PROGRAM MAIN_LD
VAR	

	// ========= System Control / FSM Variables =========
	
	MainCommands 		: MainCommands_typ; 		// command struct for cycling thru the state machine
	MainState    		: MainStateMachine_enum;   	// enumeration for the Main state machine
	System				: Mediator;					// System-level control object

	// ========= Linked NC Variables & References =========
	
	Mover    			: ARRAY[1..GVL.NUM_MOVERS] OF Mover; 	// instantiation of Mover objects. Matches the number of movers on the system
	
	// ========= Objectives & Parameters =========

	ParameterSet		: MotionParameters_typ;
	
	MoverList			: ARRAY[0..GVL.NUM_MOVERLISTS-1] OF MoverList;
	PositionTrigger		: ARRAY[0..GVL.NUM_POSITIONTRIGGERS-1] OF PositionTrigger;
	Station				: ARRAY[0..GVL.NUM_STATIONS-1] OF Station;
	Track				: ARRAY[0..GVL.NUM_TRACKS] OF Track;
	Zone				: ARRAY[0..GVL.NUM_ZONES-1] OF Zone;
	
    // ========= Helper, State, & Index Variables =========
	
    i                	: UINT; 	// index variable; gets reused in various FOR loops
    n                	: UINT; 	// secondary index variable, for enabling movers
	
	// ========= Example Application Variables =========

    nextStation 			: USINT := 4;
                    	
    lowVelocity    			: LREAL := 200;  	// mm/s
    mediumVelocity 			: LREAL := 800;  	// mm/s
    highVelocity   			: LREAL := 1200; 	// mm/s
	
	StationTimer 			: ARRAY[0..GVL.NUM_STATIONS] OF TON; // timer blocks, for station dwells
	InitialParameterSet		: MotionParameters_typ;
	
	// ========= Additional Ladder Variables =========
	MS_Disabled						: BOOL;
	MS_Initializing					: BOOL;
	MS_Enabled						: BOOL;
	MS_Run							: BOOL;
	MS_Stopping						: BOOL;
	MS_Stopped						: BOOL;
	MS_Disabling					: BOOL;
	MS_Error						: BOOL;
	MS_Debug						: BOOL;
	
	MS_Enabled_StartReady			: BOOL;
	StationGroupInPosition			: BOOL;
	StationGroupMoversInPosition	: BOOL;
	Station1_TimerIn: BOOL;
END_VAR
VAR // added by the converter: edge detectors and wires of the graphical bodies
    _w1, _w2, _w3, _w4, _w5, _w6, _w7, _w8, _w9 : BOOL;
END_VAR

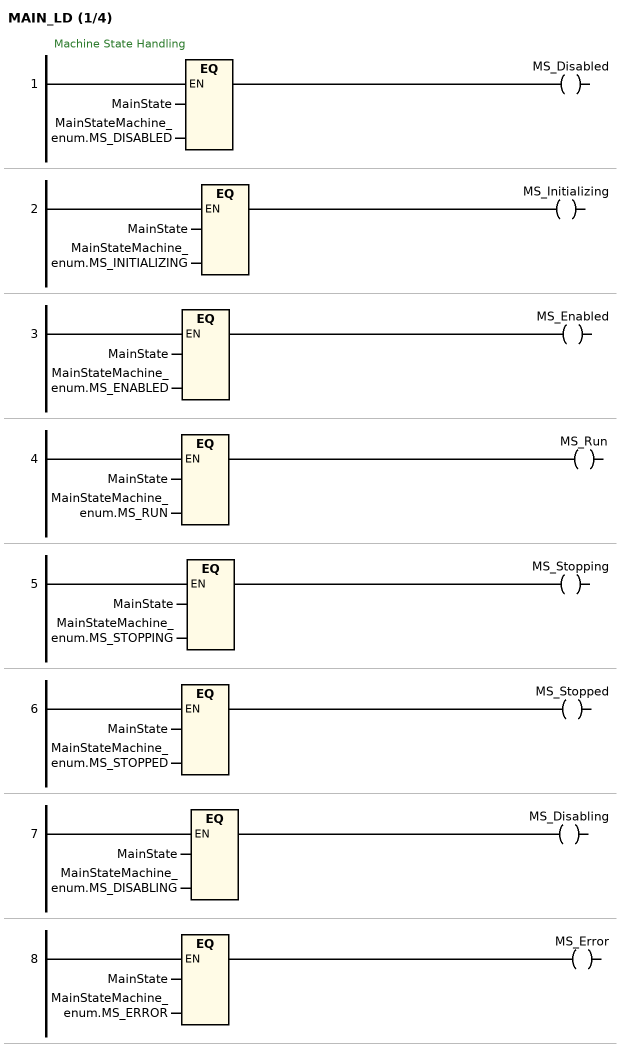
// NETWORK 1
// Machine State Handling
MS_Disabled := MainState = MainStateMachine_enum.MS_DISABLED;

// NETWORK 2
MS_Initializing := MainState = MainStateMachine_enum.MS_INITIALIZING;

// NETWORK 3
MS_Enabled := MainState = MainStateMachine_enum.MS_ENABLED;

// NETWORK 4
MS_Run := MainState = MainStateMachine_enum.MS_RUN;

// NETWORK 5
MS_Stopping := MainState = MainStateMachine_enum.MS_STOPPING;

// NETWORK 6
MS_Stopped := MainState = MainStateMachine_enum.MS_STOPPED;

// NETWORK 7
MS_Disabling := MainState = MainStateMachine_enum.MS_DISABLING;

// NETWORK 8
MS_Error := MainState = MainStateMachine_enum.MS_ERROR;

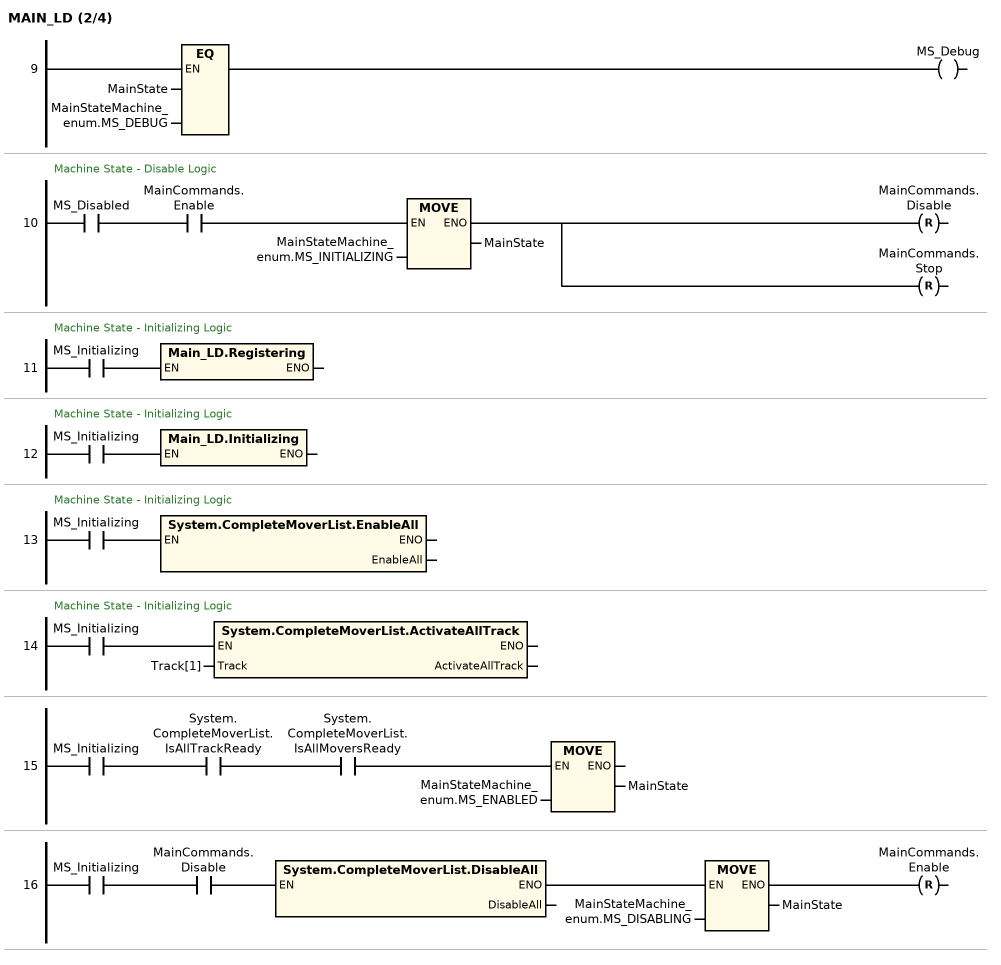
// NETWORK 9
MS_Debug := MainState = MainStateMachine_enum.MS_DEBUG;

// NETWORK 10
// Machine State - Disable Logic
_w1 := MS_Disabled AND MainCommands.Enable;
IF _w1 THEN MainState := MainStateMachine_enum.MS_INITIALIZING; END_IF
MainCommands.Disable R= _w1;
MainCommands.Stop R= _w1;

// NETWORK 11
// Machine State - Initializing Logic
IF MS_Initializing THEN Main_LD.Registering(); END_IF

// NETWORK 12
// Machine State - Initializing Logic
IF MS_Initializing THEN Main_LD.Initializing(); END_IF

// NETWORK 13
// Machine State - Initializing Logic
IF MS_Initializing THEN System.CompleteMoverList.EnableAll(); END_IF

// NETWORK 14
// Machine State - Initializing Logic
IF MS_Initializing THEN System.CompleteMoverList.ActivateAllTrack(Track := Track[1]); END_IF

// NETWORK 15
IF MS_Initializing AND System.CompleteMoverList.IsAllTrackReady AND System.CompleteMoverList.IsAllMoversReady THEN
    MainState := MainStateMachine_enum.MS_ENABLED;
END_IF

// NETWORK 16
_w2 := MS_Initializing AND MainCommands.Disable;
IF _w2 THEN System.CompleteMoverList.DisableAll(); END_IF
IF _w2 THEN MainState := MainStateMachine_enum.MS_DISABLING; END_IF
MainCommands.Enable R= _w2;

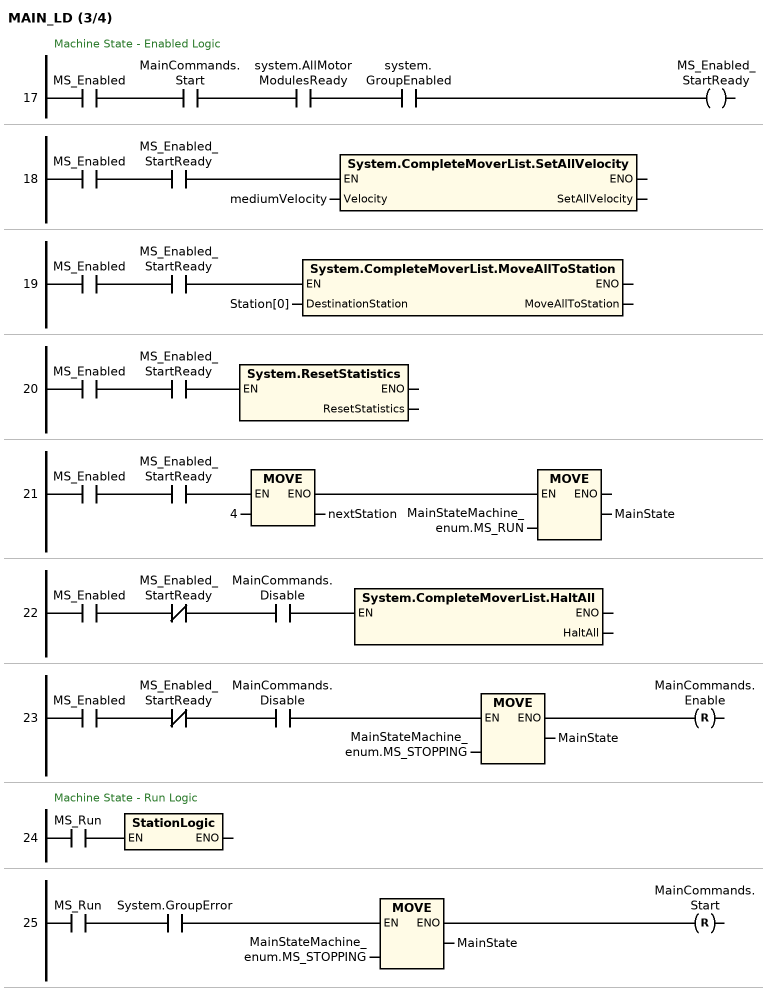
// NETWORK 17
// Machine State - Enabled Logic
MS_Enabled_StartReady := MS_Enabled AND MainCommands.Start AND system.AllMotorModulesReady AND system.GroupEnabled;

// NETWORK 18
IF MS_Enabled AND MS_Enabled_StartReady THEN
    System.CompleteMoverList.SetAllVelocity(Velocity := mediumVelocity);
END_IF

// NETWORK 19
IF MS_Enabled AND MS_Enabled_StartReady THEN
    System.CompleteMoverList.MoveAllToStation(DestinationStation := Station[0]);
END_IF

// NETWORK 20
IF MS_Enabled AND MS_Enabled_StartReady THEN System.ResetStatistics(); END_IF

// NETWORK 21
_w3 := MS_Enabled AND MS_Enabled_StartReady;
IF _w3 THEN nextStation := 4; END_IF
IF _w3 THEN MainState := MainStateMachine_enum.MS_RUN; END_IF

// NETWORK 22
IF MS_Enabled AND NOT MS_Enabled_StartReady AND MainCommands.Disable THEN
    System.CompleteMoverList.HaltAll();
END_IF

// NETWORK 23
_w4 := MS_Enabled AND NOT MS_Enabled_StartReady AND MainCommands.Disable;
IF _w4 THEN MainState := MainStateMachine_enum.MS_STOPPING; END_IF
MainCommands.Enable R= _w4;

// NETWORK 24
// Machine State - Run Logic
IF MS_Run THEN StationLogic(); END_IF

// NETWORK 25
_w5 := MS_Run AND System.GroupError;
IF _w5 THEN MainState := MainStateMachine_enum.MS_STOPPING; END_IF
MainCommands.Start R= _w5;

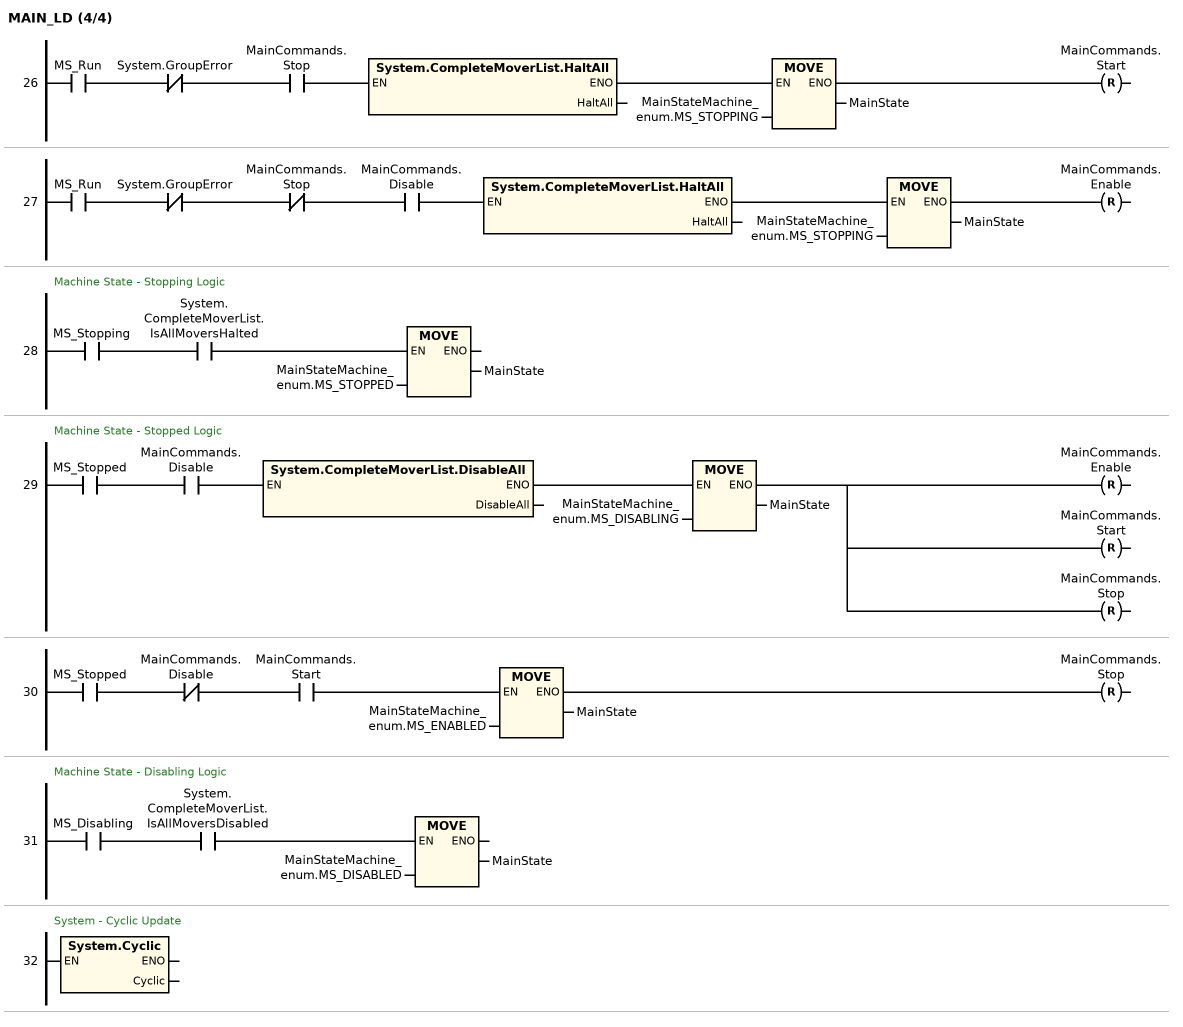
// NETWORK 26
_w6 := MS_Run AND NOT System.GroupError AND MainCommands.Stop;
IF _w6 THEN System.CompleteMoverList.HaltAll(); END_IF
IF _w6 THEN MainState := MainStateMachine_enum.MS_STOPPING; END_IF
MainCommands.Start R= _w6;

// NETWORK 27
_w7 := MS_Run AND NOT System.GroupError AND NOT MainCommands.Stop AND MainCommands.Disable;
IF _w7 THEN System.CompleteMoverList.HaltAll(); END_IF
IF _w7 THEN MainState := MainStateMachine_enum.MS_STOPPING; END_IF
MainCommands.Enable R= _w7;

// NETWORK 28
// Machine State - Stopping Logic
IF MS_Stopping AND System.CompleteMoverList.IsAllMoversHalted THEN
    MainState := MainStateMachine_enum.MS_STOPPED;
END_IF

// NETWORK 29
// Machine State - Stopped Logic
_w8 := MS_Stopped AND MainCommands.Disable;
IF _w8 THEN System.CompleteMoverList.DisableAll(); END_IF
IF _w8 THEN MainState := MainStateMachine_enum.MS_DISABLING; END_IF
MainCommands.Enable R= _w8;
MainCommands.Start R= _w8;
MainCommands.Stop R= _w8;

// NETWORK 30
_w9 := MS_Stopped AND NOT MainCommands.Disable AND MainCommands.Start;
IF _w9 THEN MainState := MainStateMachine_enum.MS_ENABLED; END_IF
MainCommands.Stop R= _w9;

// NETWORK 31
// Machine State - Disabling Logic
IF MS_Disabling AND System.CompleteMoverList.IsAllMoversDisabled THEN
    MainState := MainStateMachine_enum.MS_DISABLED;
END_IF

// NETWORK 32
// System - Cyclic Update
System.Cyclic();

ACTION Initializing:


	// Initialize station positions
	Station[0].Position 		:= 5;
	Station[1].Position 		:= 750;
	Station[2].Position 		:= 1200;
	Station[3].Position 		:= 1300;
	Station[4].Position 		:= 1400;

	PositionTrigger[0].Position := 1500;
	PositionTrigger[1].Position := 2000;
	PositionTrigger[2].Position := 3500;

	Zone[0].StartPosition		:= 3750;
	Zone[0].EndPosition   		:= 750;

	Zone[1].StartPosition 		:= 750;
	Zone[1].EndPosition   		:= 1750;

	Zone[2].StartPosition 		:= 1750;
	Zone[2].EndPosition   		:= 2750;

	Zone[3].StartPosition		:= 2750;
	Zone[3].EndPosition   		:= 3750;

	InitialParameterSet.Velocity		:= 1000;		// mm/s
	InitialParameterSet.Acceleration	:= 10_000;		// mm/s2
	InitialParameterSet.Deceleration	:= 10_000;		// mm/s2
	InitialParameterSet.Jerk			:= 100_000;		// mm/s3
	InitialParameterSet.Gap				:= 85;			// mm
	InitialParameterSet.Direction		:= mcDirectionPositive;	
	
	System.CompleteMoverList.ApplyAllParameterSet( InitialParameterSet );
END_ACTION

ACTION Registering:
	

		// Add all Movers to the Mediator
		FOR i := 1 TO GVL.NUM_MOVERS DO
			System.AddMover( Mover[i] );
		END_FOR
	
		// Add all Mover Lists to the Mediator
		FOR i := 0 TO GVL.NUM_MOVERLISTS - 1 DO
			System.AddMoverList( MoverList[i] );
		END_FOR
		
		// Add all PositionTriggers to the Mediator
		FOR i := 0 TO GVL.NUM_POSITIONTRIGGERS - 1 DO
			System.AddPositionTrigger( PositionTrigger[i] );
		END_FOR
		
		// Add all Stations to the Mediator
		FOR i := 0 TO GVL.NUM_STATIONS - 1 DO
			System.AddStation( Station[i] );
		END_FOR
		
		// Add all Tracks to the Mediator
		// note track zero is a special case, so the loop is one larger than the rest of the initalization loops
		FOR i := 0 TO GVL.NUM_TRACKS DO
			Track[i].Id := UINT_TO_INT(i);
			System.AddTrack( Track[i] );
		END_FOR
		
		// Add all Zones to the Mediator
		FOR i := 0 TO GVL.NUM_ZONES - 1 DO
			System.AddZone( Zone[i] );
		END_FOR
END_ACTION

ACTION StationLogic:
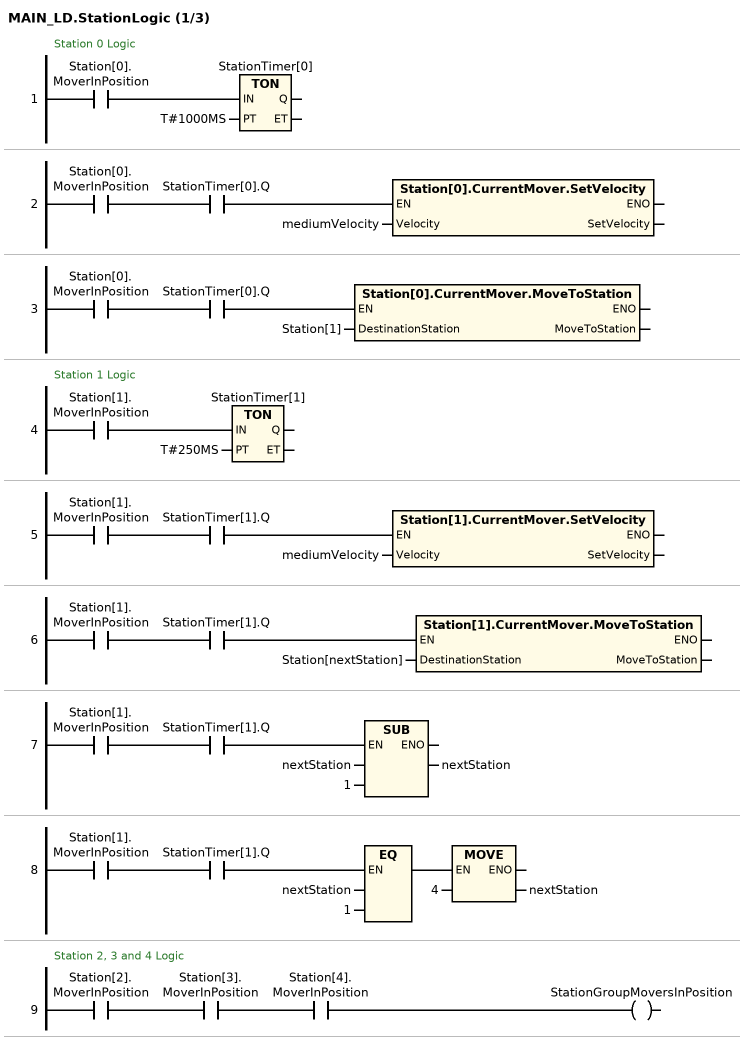
// NETWORK 1
// Station 0 Logic
StationTimer[0](IN := Station[0].MoverInPosition, PT := T#1000MS); // TON

// NETWORK 2
IF Station[0].MoverInPosition AND StationTimer[0].Q THEN
    Station[0].CurrentMover.SetVelocity(Velocity := mediumVelocity);
END_IF

// NETWORK 3
IF Station[0].MoverInPosition AND StationTimer[0].Q THEN
    Station[0].CurrentMover.MoveToStation(DestinationStation := Station[1]);
END_IF

// NETWORK 4
// Station 1 Logic
StationTimer[1](IN := Station[1].MoverInPosition, PT := T#250MS); // TON

// NETWORK 5
IF Station[1].MoverInPosition AND StationTimer[1].Q THEN
    Station[1].CurrentMover.SetVelocity(Velocity := mediumVelocity);
END_IF

// NETWORK 6
IF Station[1].MoverInPosition AND StationTimer[1].Q THEN
    Station[1].CurrentMover.MoveToStation(DestinationStation := Station[nextStation]);
END_IF

// NETWORK 7
IF Station[1].MoverInPosition AND StationTimer[1].Q THEN nextStation := nextStation - 1; END_IF

// NETWORK 8
IF Station[1].MoverInPosition AND StationTimer[1].Q AND nextStation = 1 THEN nextStation := 4; END_IF

// NETWORK 9
// Station 2, 3 and 4 Logic
StationGroupMoversInPosition := Station[2].MoverInPosition AND Station[3].MoverInPosition AND Station[4].MoverInPosition;

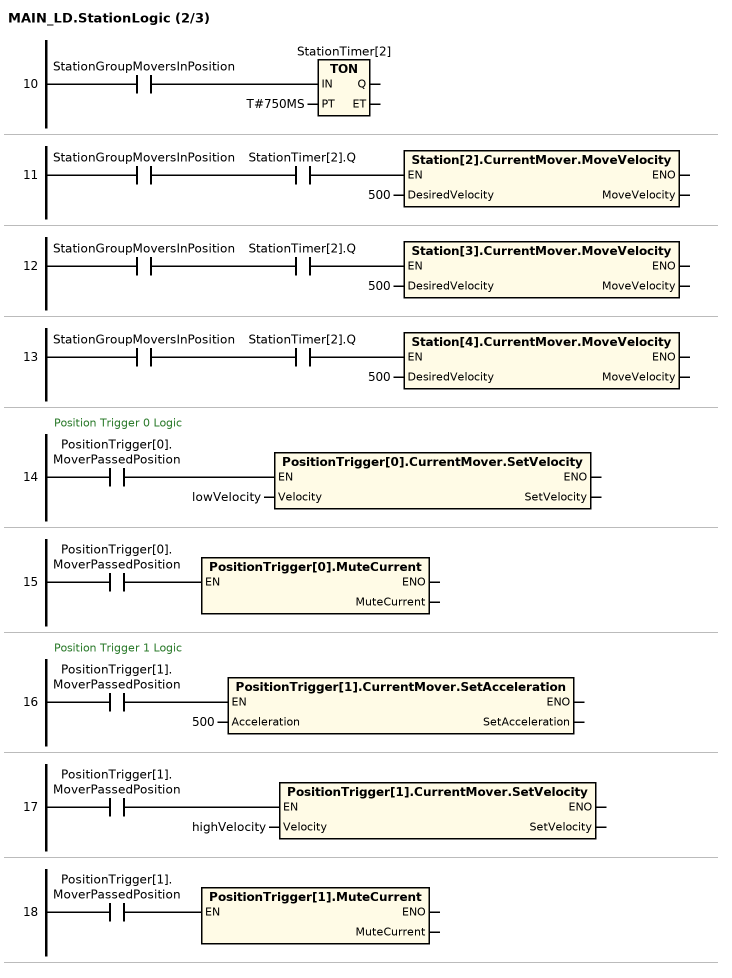
// NETWORK 10
StationTimer[2](IN := StationGroupMoversInPosition, PT := T#750MS); // TON

// NETWORK 11
IF StationGroupMoversInPosition AND StationTimer[2].Q THEN
    Station[2].CurrentMover.MoveVelocity(DesiredVelocity := 500);
END_IF

// NETWORK 12
IF StationGroupMoversInPosition AND StationTimer[2].Q THEN
    Station[3].CurrentMover.MoveVelocity(DesiredVelocity := 500);
END_IF

// NETWORK 13
IF StationGroupMoversInPosition AND StationTimer[2].Q THEN
    Station[4].CurrentMover.MoveVelocity(DesiredVelocity := 500);
END_IF

// NETWORK 14
// Position Trigger 0 Logic
IF PositionTrigger[0].MoverPassedPosition THEN
    PositionTrigger[0].CurrentMover.SetVelocity(Velocity := lowVelocity);
END_IF

// NETWORK 15
IF PositionTrigger[0].MoverPassedPosition THEN PositionTrigger[0].MuteCurrent(); END_IF

// NETWORK 16
// Position Trigger 1 Logic
IF PositionTrigger[1].MoverPassedPosition THEN
    PositionTrigger[1].CurrentMover.SetAcceleration(Acceleration := 500);
END_IF

// NETWORK 17
IF PositionTrigger[1].MoverPassedPosition THEN
    PositionTrigger[1].CurrentMover.SetVelocity(Velocity := highVelocity);
END_IF

// NETWORK 18
IF PositionTrigger[1].MoverPassedPosition THEN PositionTrigger[1].MuteCurrent(); END_IF

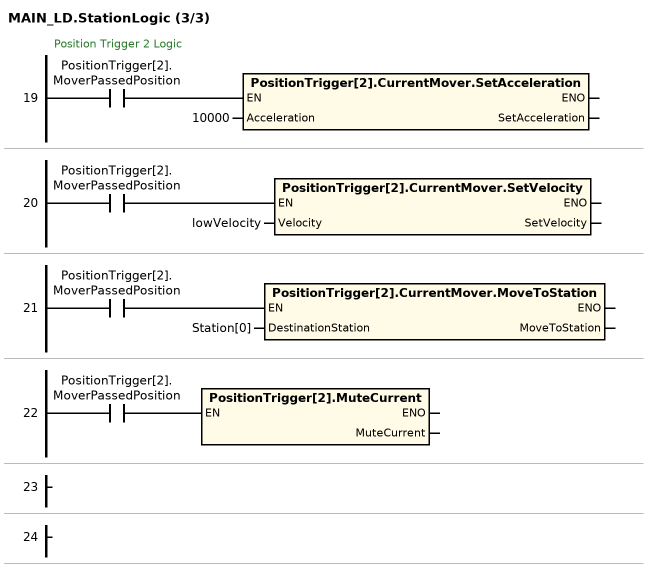
// NETWORK 19
// Position Trigger 2 Logic
IF PositionTrigger[2].MoverPassedPosition THEN
    PositionTrigger[2].CurrentMover.SetAcceleration(Acceleration := 10000);
END_IF

// NETWORK 20
IF PositionTrigger[2].MoverPassedPosition THEN
    PositionTrigger[2].CurrentMover.SetVelocity(Velocity := lowVelocity);
END_IF

// NETWORK 21
IF PositionTrigger[2].MoverPassedPosition THEN
    PositionTrigger[2].CurrentMover.MoveToStation(DestinationStation := Station[0]);
END_IF

// NETWORK 22
IF PositionTrigger[2].MoverPassedPosition THEN PositionTrigger[2].MuteCurrent(); END_IF

// NETWORK 23

// NETWORK 24
END_ACTION

END_PROGRAM

(* stored: Version 1.1.0.1, ProductVersion 3.1.4024.13
   POU MAIN_LD: Id {4697cc62-040b-0c2c-26a5-d75e283b1a86}, SpecialFunc None
   Action Initializing: Id {6204caf6-b75e-0f65-08f7-2eef4b87ad88}
   Action Registering: Id {aee1b0d6-242d-0f99-18bc-e919201d3313}
   Action StationLogic: Id {ed11c6af-3581-0b60-3f04-f27405a74e68} *)
